// TIA Portal V18 export
FUNCTION "Flowrate FC" : Void   // FC35, LAD
{ S7_Optimized_Access := 'TRUE' }
VERSION : 0.1
// stored: AutoNumber true, IsIECCheckEnabled false, SetENOAutomatically false, UDAEnableTagReadback false
BEGIN

REGION Network 1: Pump size according to ml/l/kg
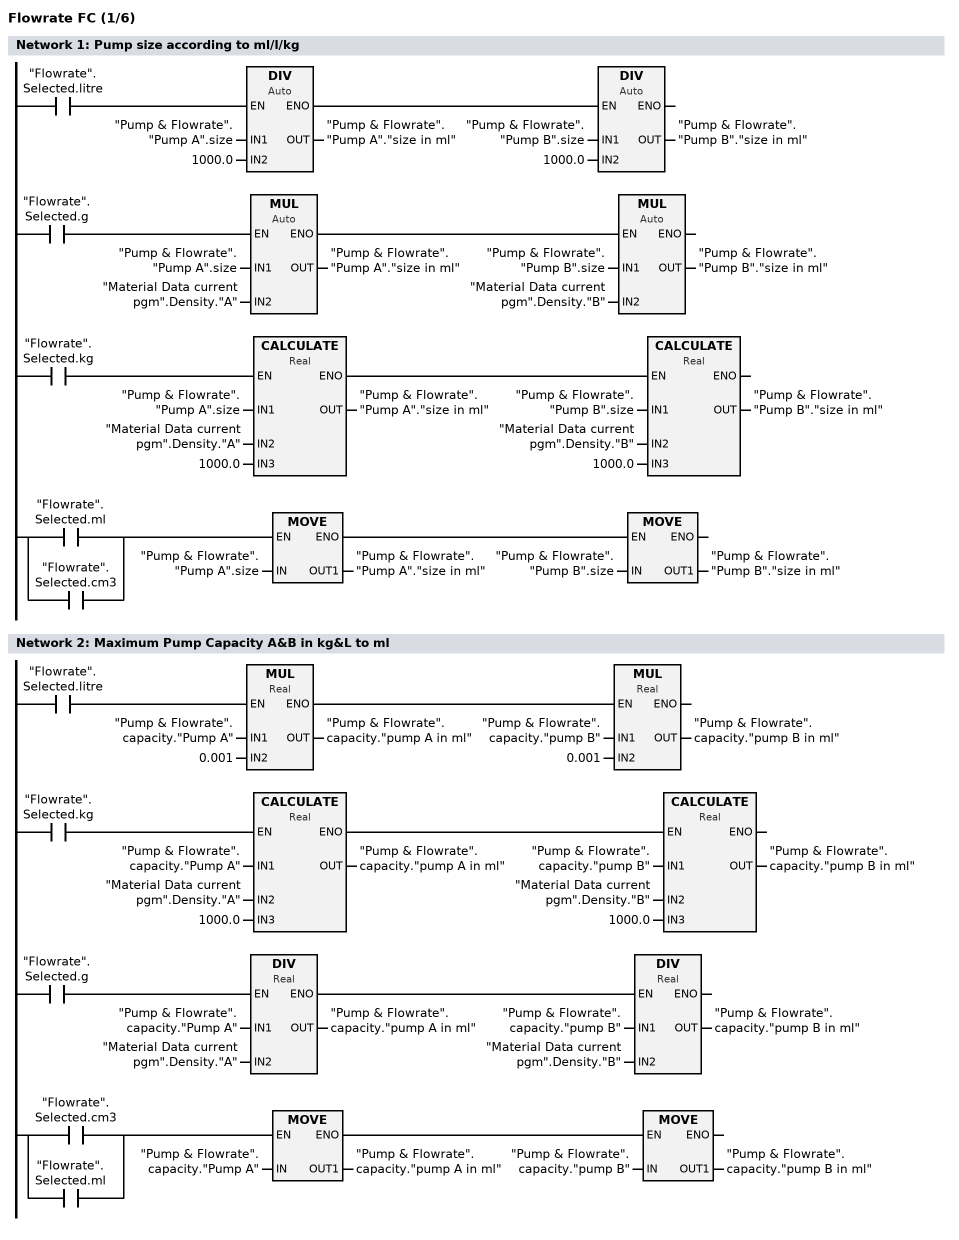
   IF "Flowrate".Selected.litre THEN
       "Pump & Flowrate"."Pump A"."size in ml" := "Pump & Flowrate"."Pump A".size / 1000.0;
       "Pump & Flowrate"."Pump B"."size in ml" := "Pump & Flowrate"."Pump B".size / 1000.0;
   END_IF;
   IF "Flowrate".Selected.g THEN
       "Pump & Flowrate"."Pump A"."size in ml" := "Pump & Flowrate"."Pump A".size * "Material Data current pgm".Density."A";
       "Pump & Flowrate"."Pump B"."size in ml" := "Pump & Flowrate"."Pump B".size * "Material Data current pgm".Density."B";
   END_IF;
   IF "Flowrate".Selected.kg THEN
       "Pump & Flowrate"."Pump A"."size in ml" := ("Pump & Flowrate"."Pump A".size*"Material Data current pgm".Density."A")/1000.0;
       "Pump & Flowrate"."Pump B"."size in ml" := ("Pump & Flowrate"."Pump B".size*"Material Data current pgm".Density."B")/1000.0;
   END_IF;
   IF "Flowrate".Selected.ml OR "Flowrate".Selected.cm3 THEN
       "Pump & Flowrate"."Pump A"."size in ml" := "Pump & Flowrate"."Pump A".size;
       "Pump & Flowrate"."Pump B"."size in ml" := "Pump & Flowrate"."Pump B".size;
   END_IF;
END_REGION

REGION Network 2: Maximum Pump Capacity A&B in kg&L to ml
   IF "Flowrate".Selected.litre THEN
       "Pump & Flowrate".capacity."pump A in ml" := "Pump & Flowrate".capacity."Pump A" * 0.001;
       "Pump & Flowrate".capacity."pump B in ml" := "Pump & Flowrate".capacity."pump B" * 0.001;
   END_IF;
   IF "Flowrate".Selected.kg THEN
       "Pump & Flowrate".capacity."pump A in ml" := ("Pump & Flowrate".capacity."Pump A"*"Material Data current pgm".Density."A")/1000.0;
       "Pump & Flowrate".capacity."pump B in ml" := ("Pump & Flowrate".capacity."pump B"*"Material Data current pgm".Density."B")/1000.0;
   END_IF;
   IF "Flowrate".Selected.g THEN
       "Pump & Flowrate".capacity."pump A in ml" := "Pump & Flowrate".capacity."Pump A" / "Material Data current pgm".Density."A";
       "Pump & Flowrate".capacity."pump B in ml" := "Pump & Flowrate".capacity."pump B" / "Material Data current pgm".Density."B";
   END_IF;
   IF "Flowrate".Selected.cm3 OR "Flowrate".Selected.ml THEN
       "Pump & Flowrate".capacity."pump A in ml" := "Pump & Flowrate".capacity."Pump A";
       "Pump & Flowrate".capacity."pump B in ml" := "Pump & Flowrate".capacity."pump B";
   END_IF;
END_REGION

REGION Network 3: Mixed flowrate Minimum
   // 10% of maximum Flowrate
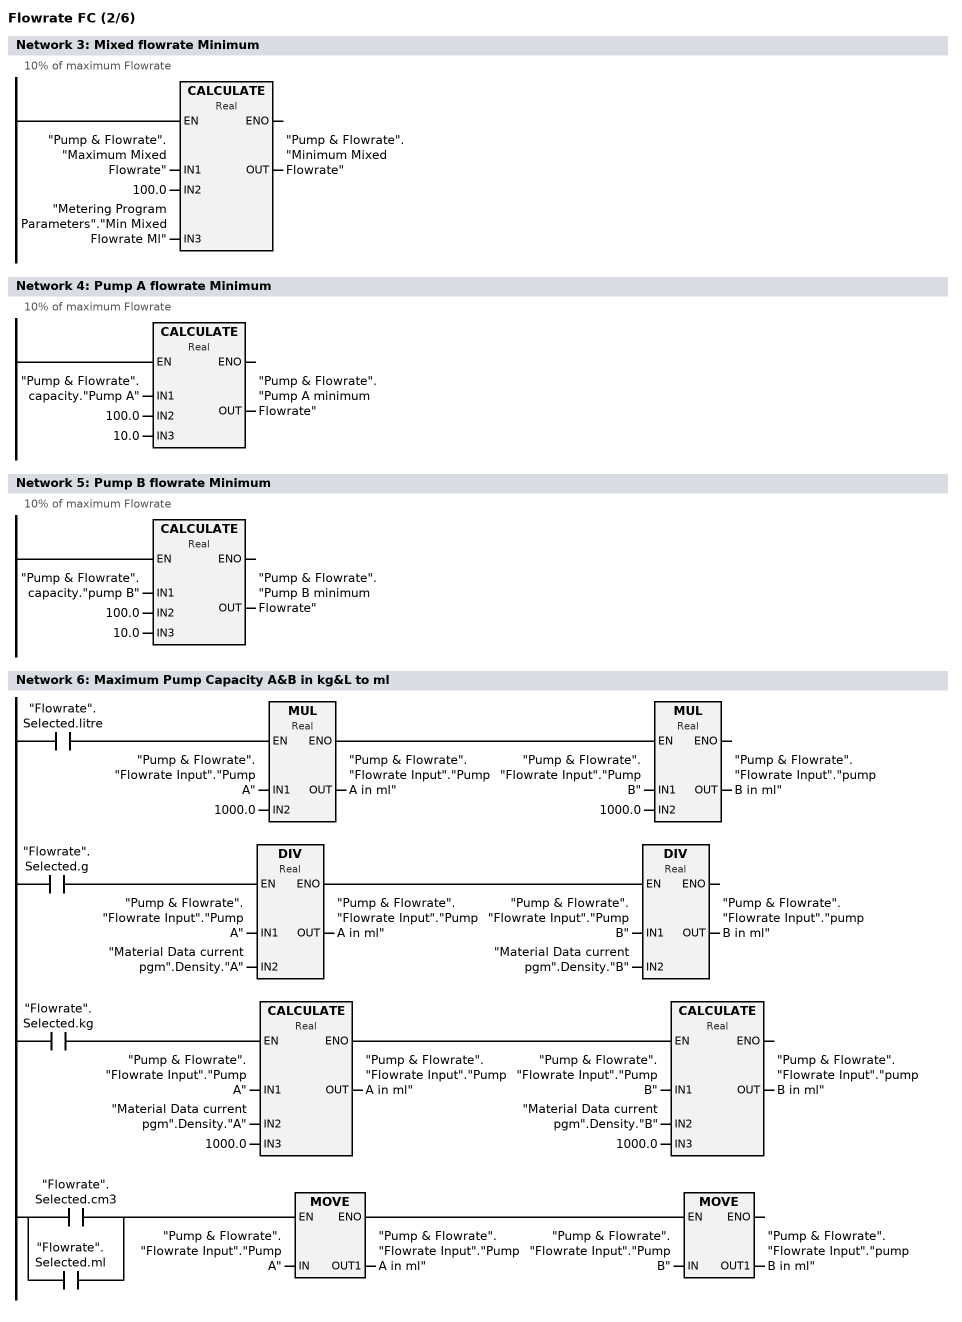
   "Pump & Flowrate"."Minimum Mixed Flowrate" := ("Pump & Flowrate"."Maximum Mixed Flowrate"/100.0)*"Metering Program Parameters"."Min Mixed Flowrate Ml";
END_REGION

REGION Network 4: Pump A flowrate Minimum
   // 10% of maximum Flowrate
   "Pump & Flowrate"."Pump A minimum Flowrate" := ("Pump & Flowrate".capacity."Pump A"/100.0)*10.0;
END_REGION

REGION Network 5: Pump B flowrate Minimum
   // 10% of maximum Flowrate
   "Pump & Flowrate"."Pump B minimum Flowrate" := ("Pump & Flowrate".capacity."pump B"/100.0)*10.0;
END_REGION

REGION Network 6: Maximum Pump Capacity A&B in kg&L to ml
   IF "Flowrate".Selected.litre THEN
       "Pump & Flowrate"."Flowrate Input"."Pump A in ml" := "Pump & Flowrate"."Flowrate Input"."Pump A" * 1000.0;
       "Pump & Flowrate"."Flowrate Input"."pump B in ml" := "Pump & Flowrate"."Flowrate Input"."Pump B" * 1000.0;
   END_IF;
   IF "Flowrate".Selected.g THEN
       "Pump & Flowrate"."Flowrate Input"."Pump A in ml" := "Pump & Flowrate"."Flowrate Input"."Pump A" / "Material Data current pgm".Density."A";
       "Pump & Flowrate"."Flowrate Input"."pump B in ml" := "Pump & Flowrate"."Flowrate Input"."Pump B" / "Material Data current pgm".Density."B";
   END_IF;
   IF "Flowrate".Selected.kg THEN
       "Pump & Flowrate"."Flowrate Input"."Pump A in ml" := ("Pump & Flowrate"."Flowrate Input"."Pump A"*"Material Data current pgm".Density."A")/1000.0;
       "Pump & Flowrate"."Flowrate Input"."pump B in ml" := ("Pump & Flowrate"."Flowrate Input"."Pump B"*"Material Data current pgm".Density."B")/1000.0;
   END_IF;
   IF "Flowrate".Selected.cm3 OR "Flowrate".Selected.ml THEN
       "Pump & Flowrate"."Flowrate Input"."Pump A in ml" := "Pump & Flowrate"."Flowrate Input"."Pump A";
       "Pump & Flowrate"."Flowrate Input"."pump B in ml" := "Pump & Flowrate"."Flowrate Input"."Pump B";
   END_IF;
END_REGION

REGION Network 7: Current Flowrate A In ml/litre/kg
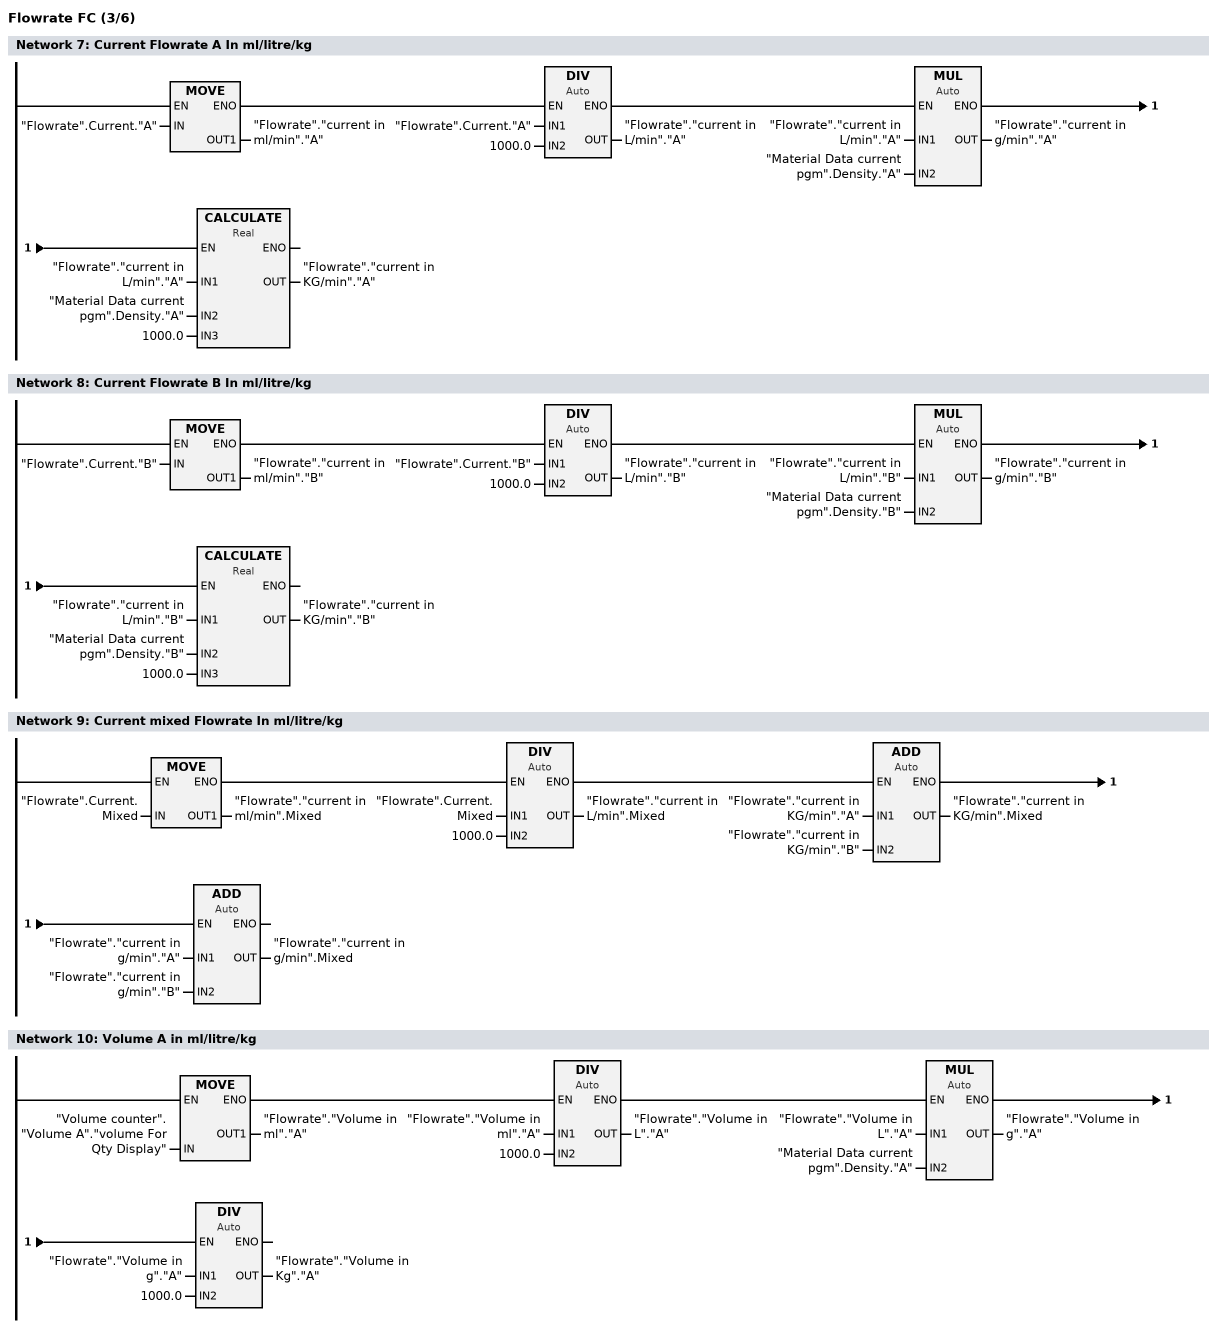
   RUNG wire#powerrail
      Move(in := "Flowrate".Current."A", out1 => "Flowrate"."current in ml/min"."A")
      Div(in1 := "Flowrate".Current."A", in2 := 1000.0, out => "Flowrate"."current in L/min"."A")
      Mul(in1 := "Flowrate"."current in L/min"."A", in2 := "Material Data current pgm".Density."A", out => "Flowrate"."current in g/min"."A")
      { S7_Templates := "SrcType := Real"; S7_Expression := "(IN1*IN2)/IN3" } Calculate(in1 := "Flowrate"."current in L/min"."A", in2 := "Material Data current pgm".Density."A", in3 := 1000.0, out => "Flowrate"."current in KG/min"."A")
   END_RUNG
   // the same network as SCL:
   "Flowrate"."current in ml/min"."A" := "Flowrate".Current."A";
   "Flowrate"."current in L/min"."A" := "Flowrate".Current."A" / 1000.0;
   "Flowrate"."current in g/min"."A" := "Flowrate"."current in L/min"."A" * "Material Data current pgm".Density."A";
   "Flowrate"."current in KG/min"."A" := ("Flowrate"."current in L/min"."A"*"Material Data current pgm".Density."A")/1000.0;
END_REGION

REGION Network 8: Current Flowrate B In ml/litre/kg
   RUNG wire#powerrail
      Move(in := "Flowrate".Current."B", out1 => "Flowrate"."current in ml/min"."B")
      Div(in1 := "Flowrate".Current."B", in2 := 1000.0, out => "Flowrate"."current in L/min"."B")
      Mul(in1 := "Flowrate"."current in L/min"."B", in2 := "Material Data current pgm".Density."B", out => "Flowrate"."current in g/min"."B")
      { S7_Templates := "SrcType := Real"; S7_Expression := "(IN1*IN2)/IN3" } Calculate(in1 := "Flowrate"."current in L/min"."B", in2 := "Material Data current pgm".Density."B", in3 := 1000.0, out => "Flowrate"."current in KG/min"."B")
   END_RUNG
   // the same network as SCL:
   "Flowrate"."current in ml/min"."B" := "Flowrate".Current."B";
   "Flowrate"."current in L/min"."B" := "Flowrate".Current."B" / 1000.0;
   "Flowrate"."current in g/min"."B" := "Flowrate"."current in L/min"."B" * "Material Data current pgm".Density."B";
   "Flowrate"."current in KG/min"."B" := ("Flowrate"."current in L/min"."B"*"Material Data current pgm".Density."B")/1000.0;
END_REGION

REGION Network 9: Current mixed Flowrate In ml/litre/kg
   RUNG wire#powerrail
      Move(in := "Flowrate".Current.Mixed, out1 => "Flowrate"."current in ml/min".Mixed)
      Div(in1 := "Flowrate".Current.Mixed, in2 := 1000.0, out => "Flowrate"."current in L/min".Mixed)
      Add(in1 := "Flowrate"."current in KG/min"."A", in2 := "Flowrate"."current in KG/min"."B", out => "Flowrate"."current in KG/min".Mixed)
      Add(in1 := "Flowrate"."current in g/min"."A", in2 := "Flowrate"."current in g/min"."B", out => "Flowrate"."current in g/min".Mixed)
   END_RUNG
   // the same network as SCL:
   "Flowrate"."current in ml/min".Mixed := "Flowrate".Current.Mixed;
   "Flowrate"."current in L/min".Mixed := "Flowrate".Current.Mixed / 1000.0;
   "Flowrate"."current in KG/min".Mixed := "Flowrate"."current in KG/min"."A" + "Flowrate"."current in KG/min"."B";
   "Flowrate"."current in g/min".Mixed := "Flowrate"."current in g/min"."A" + "Flowrate"."current in g/min"."B";
END_REGION

REGION Network 10: Volume A in ml/litre/kg
   RUNG wire#powerrail
      Move(in := "Volume counter"."Volume A"."volume For Qty Display", out1 => "Flowrate"."Volume in ml"."A")
      Div(in1 := "Flowrate"."Volume in ml"."A", in2 := 1000.0, out => "Flowrate"."Volume in L"."A")
      Mul(in1 := "Flowrate"."Volume in L"."A", in2 := "Material Data current pgm".Density."A", out => "Flowrate"."Volume in g"."A")
      Div(in1 := "Flowrate"."Volume in g"."A", in2 := 1000.0, out => "Flowrate"."Volume in Kg"."A")
   END_RUNG
   // the same network as SCL:
   "Flowrate"."Volume in ml"."A" := "Volume counter"."Volume A"."volume For Qty Display";
   "Flowrate"."Volume in L"."A" := "Flowrate"."Volume in ml"."A" / 1000.0;
   "Flowrate"."Volume in g"."A" := "Flowrate"."Volume in L"."A" * "Material Data current pgm".Density."A";
   "Flowrate"."Volume in Kg"."A" := "Flowrate"."Volume in g"."A" / 1000.0;
END_REGION

REGION Network 11: Volume B in ml/litre/kg
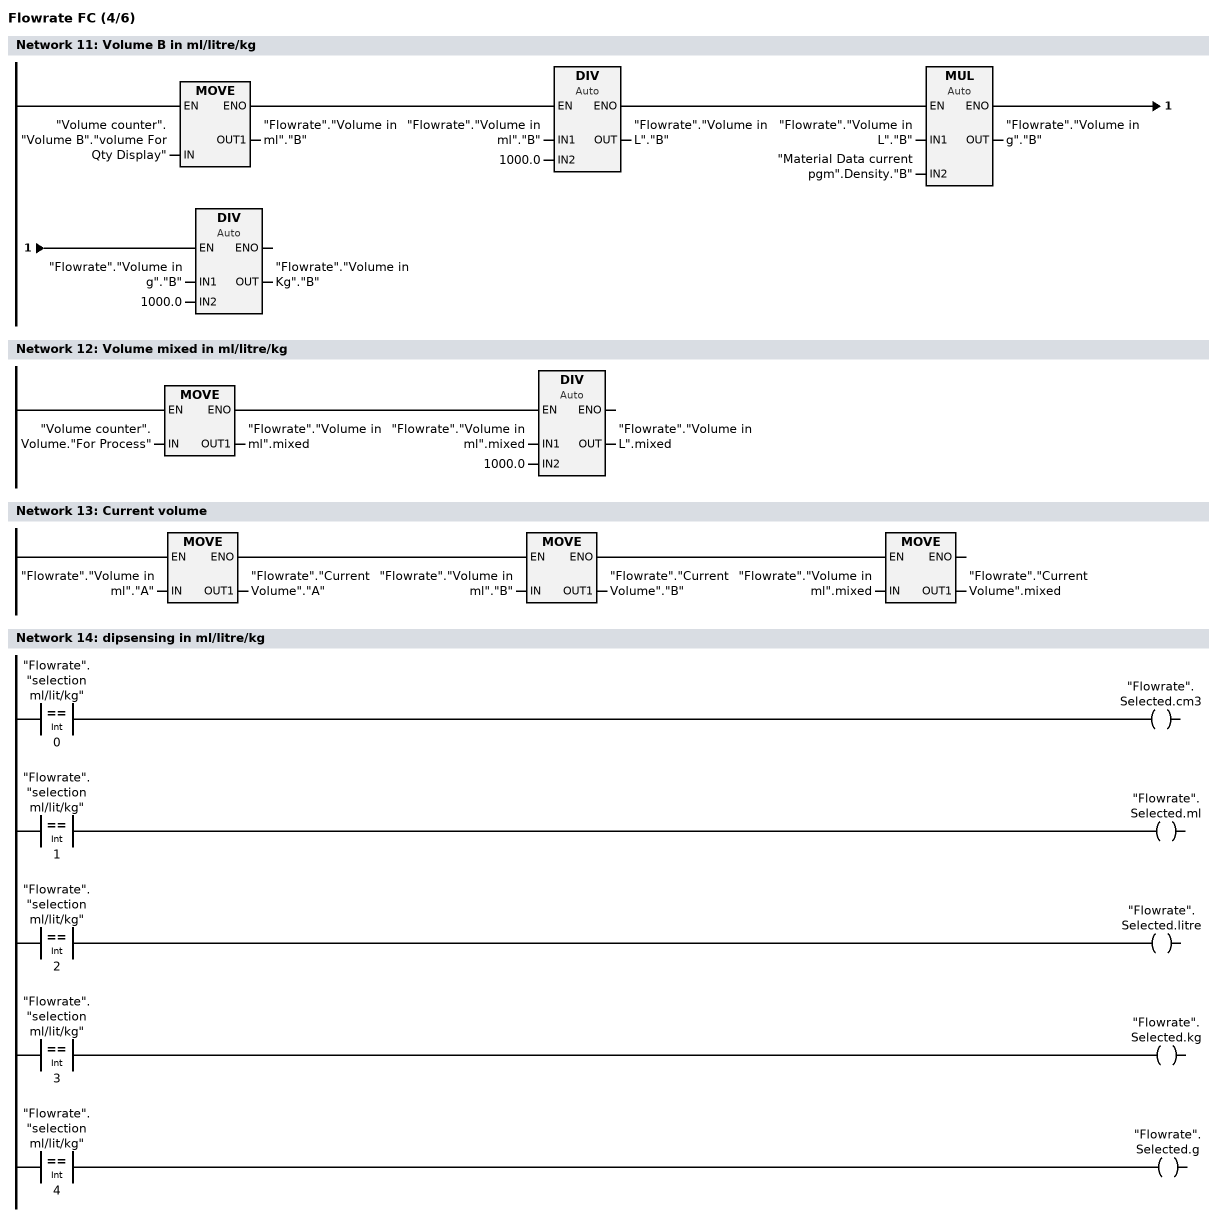
   RUNG wire#powerrail
      Move(in := "Volume counter"."Volume B"."volume For Qty Display", out1 => "Flowrate"."Volume in ml"."B")
      Div(in1 := "Flowrate"."Volume in ml"."B", in2 := 1000.0, out => "Flowrate"."Volume in L"."B")
      Mul(in1 := "Flowrate"."Volume in L"."B", in2 := "Material Data current pgm".Density."B", out => "Flowrate"."Volume in g"."B")
      Div(in1 := "Flowrate"."Volume in g"."B", in2 := 1000.0, out => "Flowrate"."Volume in Kg"."B")
   END_RUNG
   // the same network as SCL:
   "Flowrate"."Volume in ml"."B" := "Volume counter"."Volume B"."volume For Qty Display";
   "Flowrate"."Volume in L"."B" := "Flowrate"."Volume in ml"."B" / 1000.0;
   "Flowrate"."Volume in g"."B" := "Flowrate"."Volume in L"."B" * "Material Data current pgm".Density."B";
   "Flowrate"."Volume in Kg"."B" := "Flowrate"."Volume in g"."B" / 1000.0;
END_REGION

REGION Network 12: Volume mixed in ml/litre/kg
   RUNG wire#powerrail
      Move(in := "Volume counter".Volume."For Process", out1 => "Flowrate"."Volume in ml".mixed)
      Div(in1 := "Flowrate"."Volume in ml".mixed, in2 := 1000.0, out => "Flowrate"."Volume in L".mixed)
   END_RUNG
   // the same network as SCL:
   "Flowrate"."Volume in ml".mixed := "Volume counter".Volume."For Process";
   "Flowrate"."Volume in L".mixed := "Flowrate"."Volume in ml".mixed / 1000.0;
END_REGION

REGION Network 13: Current volume
   RUNG wire#powerrail
      Move(in := "Flowrate"."Volume in ml"."A", out1 => "Flowrate"."Current Volume"."A")
      Move(in := "Flowrate"."Volume in ml"."B", out1 => "Flowrate"."Current Volume"."B")
      Move(in := "Flowrate"."Volume in ml".mixed, out1 => "Flowrate"."Current Volume".mixed)
   END_RUNG
   // the same network as SCL:
   "Flowrate"."Current Volume"."A" := "Flowrate"."Volume in ml"."A";
   "Flowrate"."Current Volume"."B" := "Flowrate"."Volume in ml"."B";
   "Flowrate"."Current Volume".mixed := "Flowrate"."Volume in ml".mixed;
END_REGION

REGION Network 14: dipsensing in ml/litre/kg
   RUNG wire#powerrail
      { S7_Templates := "SrcType := Int" } EQ_Contact(in1 := "Flowrate"."selection ml/lit/kg", in2 := 0)
      Coil( "Flowrate".Selected.cm3 )
   END_RUNG
   RUNG wire#powerrail
      { S7_Templates := "SrcType := Int" } EQ_Contact(in1 := "Flowrate"."selection ml/lit/kg", in2 := 1)
      Coil( "Flowrate".Selected.ml )
   END_RUNG
   RUNG wire#powerrail
      { S7_Templates := "SrcType := Int" } EQ_Contact(in1 := "Flowrate"."selection ml/lit/kg", in2 := 2)
      Coil( "Flowrate".Selected.litre )
   END_RUNG
   RUNG wire#powerrail
      { S7_Templates := "SrcType := Int" } EQ_Contact(in1 := "Flowrate"."selection ml/lit/kg", in2 := 3)
      Coil( "Flowrate".Selected.kg )
   END_RUNG
   RUNG wire#powerrail
      { S7_Templates := "SrcType := Int" } EQ_Contact(in1 := "Flowrate"."selection ml/lit/kg", in2 := 4)
      Coil( "Flowrate".Selected.g )
   END_RUNG
   // the same network as SCL:
   "Flowrate".Selected.cm3 := "Flowrate"."selection ml/lit/kg" = 0;
   "Flowrate".Selected.ml := "Flowrate"."selection ml/lit/kg" = 1;
   "Flowrate".Selected.litre := "Flowrate"."selection ml/lit/kg" = 2;
   "Flowrate".Selected.kg := "Flowrate"."selection ml/lit/kg" = 3;
   "Flowrate".Selected.g := "Flowrate"."selection ml/lit/kg" = 4;
END_REGION

REGION Network 15: Display flowrate in ml
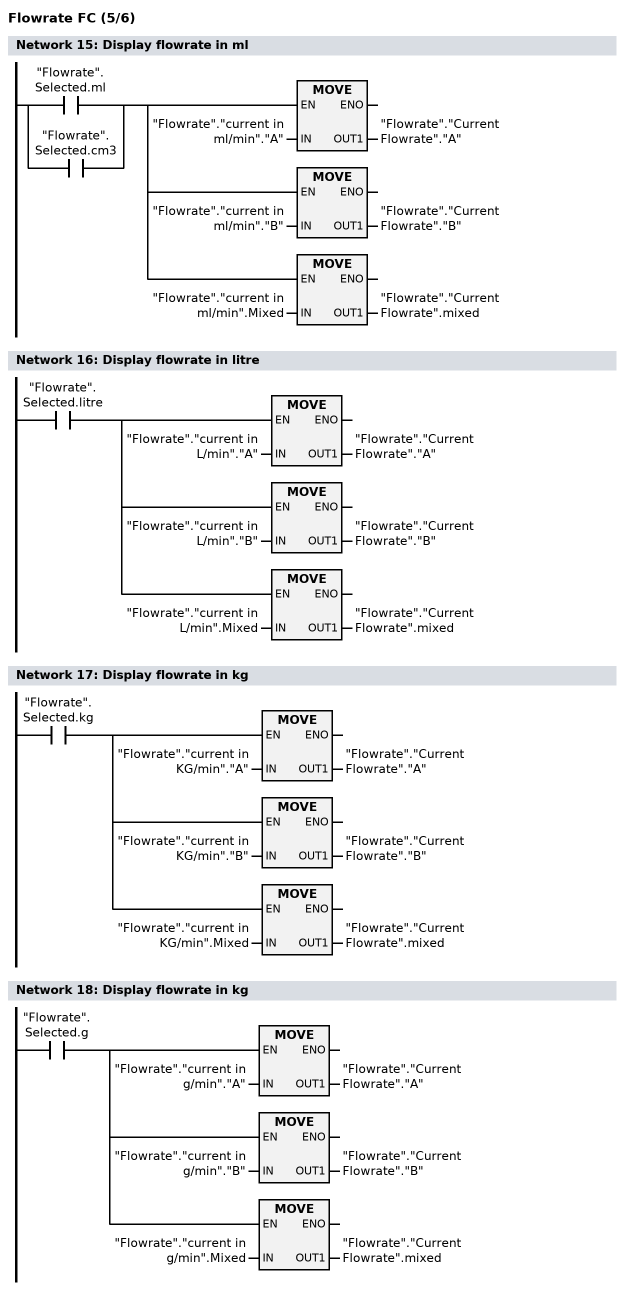
   RUNG wire#powerrail
      Contact( "Flowrate".Selected.ml )
      wire#w1
      Move(in := "Flowrate"."current in ml/min"."A", out1 => "Flowrate"."Current Flowrate"."A")
   END_RUNG
   RUNG wire#powerrail
      Contact( "Flowrate".Selected.cm3 )
   END_RUNG wire#w1
   RUNG wire#w1
      Move(in := "Flowrate"."current in ml/min"."B", out1 => "Flowrate"."Current Flowrate"."B")
   END_RUNG
   RUNG wire#w1
      Move(in := "Flowrate"."current in ml/min".Mixed, out1 => "Flowrate"."Current Flowrate".mixed)
   END_RUNG
   // the same network as SCL:
   IF "Flowrate".Selected.ml OR "Flowrate".Selected.cm3 THEN
       "Flowrate"."Current Flowrate"."A" := "Flowrate"."current in ml/min"."A";
       "Flowrate"."Current Flowrate"."B" := "Flowrate"."current in ml/min"."B";
       "Flowrate"."Current Flowrate".mixed := "Flowrate"."current in ml/min".Mixed;
   END_IF;
END_REGION

REGION Network 16: Display flowrate in litre
   RUNG wire#powerrail
      Contact( "Flowrate".Selected.litre )
      wire#w1
      Move(in := "Flowrate"."current in L/min"."A", out1 => "Flowrate"."Current Flowrate"."A")
   END_RUNG
   RUNG wire#w1
      Move(in := "Flowrate"."current in L/min"."B", out1 => "Flowrate"."Current Flowrate"."B")
   END_RUNG
   RUNG wire#w1
      Move(in := "Flowrate"."current in L/min".Mixed, out1 => "Flowrate"."Current Flowrate".mixed)
   END_RUNG
   // the same network as SCL:
   IF "Flowrate".Selected.litre THEN
       "Flowrate"."Current Flowrate"."A" := "Flowrate"."current in L/min"."A";
       "Flowrate"."Current Flowrate"."B" := "Flowrate"."current in L/min"."B";
       "Flowrate"."Current Flowrate".mixed := "Flowrate"."current in L/min".Mixed;
   END_IF;
END_REGION

REGION Network 17: Display flowrate in kg
   RUNG wire#powerrail
      Contact( "Flowrate".Selected.kg )
      wire#w1
      Move(in := "Flowrate"."current in KG/min"."A", out1 => "Flowrate"."Current Flowrate"."A")
   END_RUNG
   RUNG wire#w1
      Move(in := "Flowrate"."current in KG/min"."B", out1 => "Flowrate"."Current Flowrate"."B")
   END_RUNG
   RUNG wire#w1
      Move(in := "Flowrate"."current in KG/min".Mixed, out1 => "Flowrate"."Current Flowrate".mixed)
   END_RUNG
   // the same network as SCL:
   IF "Flowrate".Selected.kg THEN
       "Flowrate"."Current Flowrate"."A" := "Flowrate"."current in KG/min"."A";
       "Flowrate"."Current Flowrate"."B" := "Flowrate"."current in KG/min"."B";
       "Flowrate"."Current Flowrate".mixed := "Flowrate"."current in KG/min".Mixed;
   END_IF;
END_REGION

REGION Network 18: Display flowrate in kg
   RUNG wire#powerrail
      Contact( "Flowrate".Selected.g )
      wire#w1
      Move(in := "Flowrate"."current in g/min"."A", out1 => "Flowrate"."Current Flowrate"."A")
   END_RUNG
   RUNG wire#w1
      Move(in := "Flowrate"."current in g/min"."B", out1 => "Flowrate"."Current Flowrate"."B")
   END_RUNG
   RUNG wire#w1
      Move(in := "Flowrate"."current in g/min".Mixed, out1 => "Flowrate"."Current Flowrate".mixed)
   END_RUNG
   // the same network as SCL:
   IF "Flowrate".Selected.g THEN
       "Flowrate"."Current Flowrate"."A" := "Flowrate"."current in g/min"."A";
       "Flowrate"."Current Flowrate"."B" := "Flowrate"."current in g/min"."B";
       "Flowrate"."Current Flowrate".mixed := "Flowrate"."current in g/min".Mixed;
   END_IF;
END_REGION

REGION Network 19: Flowrate tolerence
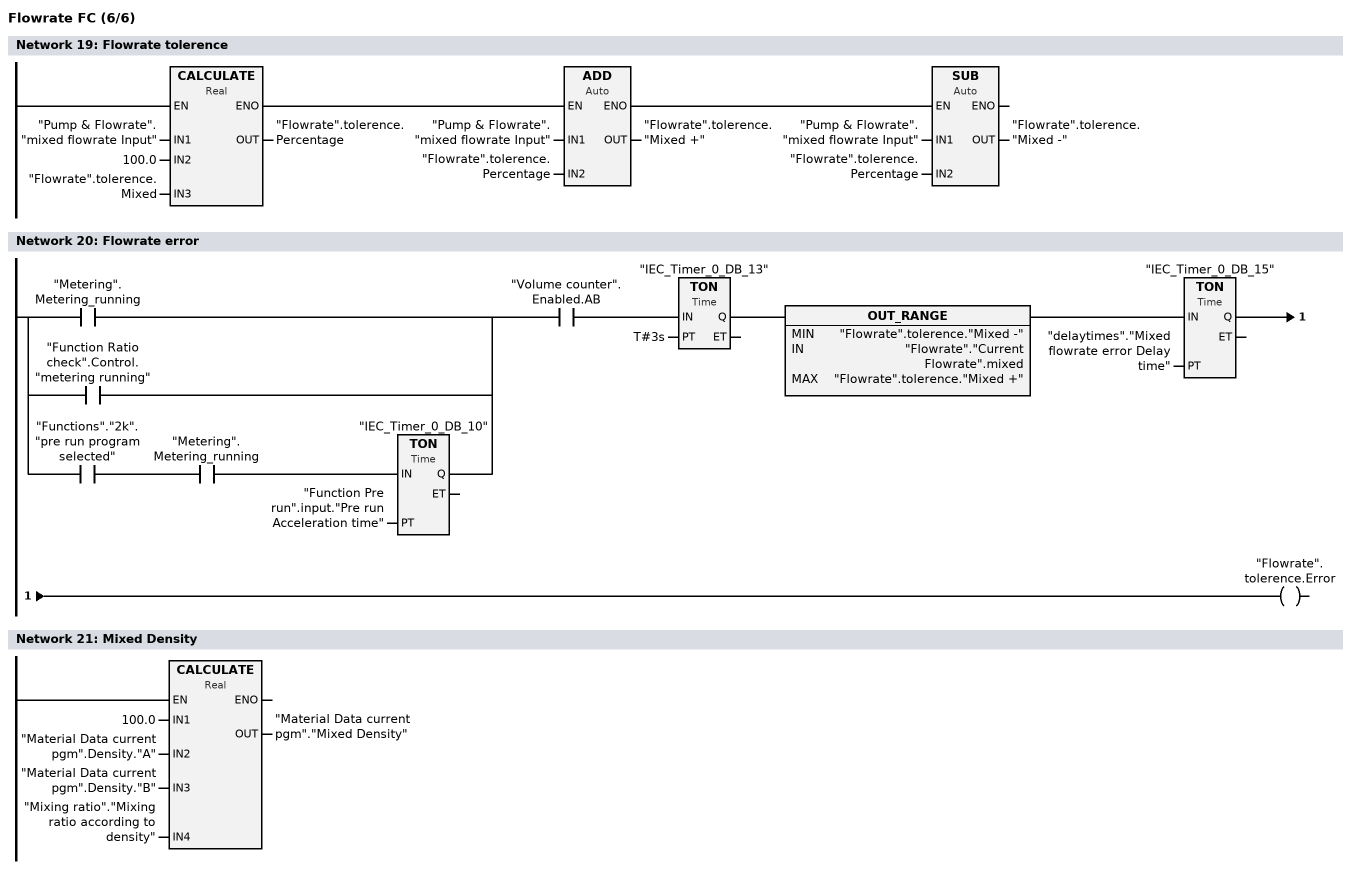
   RUNG wire#powerrail
      { S7_Templates := "SrcType := Real"; S7_Expression := "(IN1/IN2)*IN3" } Calculate(in1 := "Pump & Flowrate"."mixed flowrate Input", in2 := 100.0, in3 := "Flowrate".tolerence.Mixed, out => "Flowrate".tolerence.Percentage)
      Add(in1 := "Pump & Flowrate"."mixed flowrate Input", in2 := "Flowrate".tolerence.Percentage, out => "Flowrate".tolerence."Mixed +")
      Sub(in1 := "Pump & Flowrate"."mixed flowrate Input", in2 := "Flowrate".tolerence.Percentage, out => "Flowrate".tolerence."Mixed -")
   END_RUNG
   // the same network as SCL:
   "Flowrate".tolerence.Percentage := ("Pump & Flowrate"."mixed flowrate Input"/100.0)*"Flowrate".tolerence.Mixed;
   "Flowrate".tolerence."Mixed +" := "Pump & Flowrate"."mixed flowrate Input" + "Flowrate".tolerence.Percentage;
   "Flowrate".tolerence."Mixed -" := "Pump & Flowrate"."mixed flowrate Input" - "Flowrate".tolerence.Percentage;
END_REGION

REGION Network 20: Flowrate error
   "IEC_Timer_0_DB_10".TON(IN := "Functions"."2k"."pre run program selected" AND "Metering".Metering_running,
                           PT := "Function Pre run".input."Pre run Acceleration time");
   "IEC_Timer_0_DB_13".TON(IN := ("Metering".Metering_running OR "Function Ratio check".Control."metering running" OR "IEC_Timer_0_DB_10".Q) AND "Volume counter".Enabled.AB,
                           PT := T#3s);
   "IEC_Timer_0_DB_15".TON(IN := "IEC_Timer_0_DB_13".Q AND (("Flowrate"."Current Flowrate".mixed < "Flowrate".tolerence."Mixed -") OR ("Flowrate"."Current Flowrate".mixed > "Flowrate".tolerence."Mixed +")),
                           PT := "delaytimes"."Mixed flowrate error Delay time");
   "Flowrate".tolerence.Error := "IEC_Timer_0_DB_15".Q;
END_REGION

REGION Network 21: Mixed Density
   RUNG wire#powerrail
      { S7_Templates := "SrcType := Real"; S7_Expression := "(IN2*IN1+IN3*IN4)/(IN1+IN4)" } Calculate(in1 := 100.0, in2 := "Material Data current pgm".Density."A", in3 := "Material Data current pgm".Density."B", in4 := "Mixing ratio"."Mixing ratio according to density", out => "Material Data current pgm"."Mixed Density")
   END_RUNG
   // the same network as SCL:
   "Material Data current pgm"."Mixed Density" := ("Material Data current pgm".Density."A"*100.0+"Material Data current pgm".Density."B"*"Mixing ratio"."Mixing ratio according to density")/(100.0+"Mixing ratio"."Mixing ratio according to density");
END_REGION
END_FUNCTION
